// TIA Portal V17 export
// export: Created 2023-12-22T15:03:09.6834511Z, ExportSetting WithDefaults, DisplayName Totally Integrated Automation Portal, DisplayVersion V17, DisplayName TIA Portal Openness, DisplayVersion V17, DisplayName TIA Portal Version Control Interface, DisplayVersion V17, DisplayName STEP 7 Professional, DisplayVersion V17, DisplayName STEP 7 Safety, DisplayVersion V17, DisplayName WinCC Advanced, DisplayVersion V17
DATA_BLOCK "LE_DB"   // DB396
{ S7_Optimized_Access := 'FALSE' }
VERSION : 0.1
// stored: AutoNumber false, DBAccessibleFromOPCUA true, DBAccessibleFromWebserver true, IsOnlyStoredInLoadMemory false, IsWriteProtectedInAS false
   VAR RETAIN
      LE : Array[0..10] of Struct   // Чтение - Input Register (04), Запись - Holding Register (06)
         LE_1 : Real;   // Накопленный объем +
         LE_2 : Real;   // Накопленный объём -
         LE_3 : Real;   // Мгновенный расход
         res_2 : Real;   // Температура канала 1, С
         res_3 : Real;   // Температура канала 2, С
         res_4 : Real;   // Давление среды, кПа
         Use { S7_SetPoint := 'True'} : Bool;
         Link : Bool;
         NoRead : Bool;
         NoWrite : Bool;
         ID { S7_SetPoint := 'True'} : Int;
         ADDR { S7_SetPoint := 'True'} : UInt;
         "Name" { S7_SetPoint := 'True'} : String[10];
      END_STRUCT;
   END_VAR
BEGIN
   LE[0].Use := FALSE;
   LE[1..2].Use := TRUE;
   LE[3..10].Use := FALSE;
   LE[0].ID := 0;
   LE[1..2].ID := 14;
   LE[3..10].ID := 0;
   LE[0].ADDR := 0;
   LE[1].ADDR := 41;
   LE[2].ADDR := 42;
   LE[3..10].ADDR := 0;
   LE[0]."Name" := '';
   LE[1]."Name" := 'FE';
   LE[2..10]."Name" := '';
END_DATA_BLOCK
